Staubli VAL3: init.pgx

program init(num& x_nError[] (dimensions=1))
  local bool l_bIsScara
  local bool l_bLock
  local bool l_bQuit
  local num l_i
  local num l_nEditNR
  local num l_nError
  local num l_nRevisionNR
  local num l_nStep
  local num l_nVersionNR
  local num l_nVersionNum
  local string l_sMessage
  local string l_sSubString
begin
  //
  l_nStep=20
  l_bLock=false
  l_bQuit=false
  x_nError=0
  do
    switch l_nStep
      //Version checking
      case 0
        // Software requires VAL3 version s7.6.0 or later with valtrack license
        if l_bLock==false
          call ut:_getVersion(l_nVersionNR,l_nRevisionNR,l_nEditNR,l_nError)
          l_nVersionNum=(l_nVersionNR*100+l_nRevisionNR*10+l_nEditNR)
          l_bLock=true
          //? "version : "+toString("",l_nVersionNum)
        endIf
        if l_bLock==true
          if (l_nVersionNum>=760)
            l_nStep=10
          else
            l_nStep=50
          endIf
          l_bLock=false
        endIf
      break
      // Check if valTrack Option is installed
      case 10
        if l_bLock==false
          l_bLock=true
        endIf
        if l_bLock==true
          if getVersion("valTrack")!=""
            l_nStep=20
          else
            x_nError=47
            sErrorMessage=lang:sListOfMessage[x_nError]
            l_bQuit=true
          endIf
          l_bLock=false
        endIf
      break
      // Initialize string and tools variables
      // Load libraries
      case 20
        if l_bLock==false
          //? getVersion("ArmType")
          bIsScara=left(getVersion("ArmType"),2)=="rs"
          bIsScara=left(getVersion("ArmType"),2)=="ts" or bIsScara
          bIsScara=left(getVersion("ArmType"),2)=="tp" or bIsScara
          if bIsScara==true
            sGeometryLib=cfg:sGEOMETRYLIB_RS
          else
            sGeometryLib=cfg:sGEOMETRYLIB
          endIf
          //
          // Initialise private Tool
          tPointer.trsf=position(cfg:tPointer,flange)
          //
          // Load Geometry libray according to robot type (Scara/6axis)
          l_nError=geometry:libLoad(cfg:sPATHTEMPLATE+sGeometryLib)
          l_bLock=true
        endIf
        if l_bLock==true
          if l_nError==0
            l_nStep=30
          else
            // Prepare clear text error message
            x_nError=33
            l_sSubString=cfg:sPATHTEMPLATE+sGeometryLib
            call ut:addStrToString(lang:sListOfMessage[x_nError],sErrorMessage,"",l_sSubString)
            call ut:addNumToString(sErrorMessage,sErrorMessage,"*",l_nError)
          endIf
          l_bLock=false
        endIf
      break
      // Buil List of IOs
      case 30
        if l_bLock==false
          call buildOutputList()
          l_bLock=true
          l_bQuit=true
        endIf
      break
      // Not a valid VAL3 version
      case 50
        if l_bLock==false
          // Prepare clear text error message
          x_nError=46
          sErrorMessage=lang:sListOfMessage[x_nError]
          l_bLock=true
        endIf
        l_bQuit=true
      break
      //
    endSwitch
    delay(0)
  until (l_bQuit==true)
end
